Fanuc KAREL source: kd00015.KL

-- PROVISIONAL review KL for V940-1; original PC SHA256 e6e87a3893e7b443648327836266338668fe3b07deccfcc8bc3f06a5f374e33c
-- Incomplete behavior may be omitted. Consult companion uncertainty JSON. Do not deploy.
PROGRAM KD00015
%NOLOCKGROUP
VAR
  I : INTEGER
  J : INTEGER
  B : BOOLEAN
  R : REAL
  S : STRING[80]
BEGIN
  -- V9_ZERO_TABLE_METADATA_HINT layout=0001; no indexed target words; source/name/runtime held
  -- UNRESOLVED_PC offsets 5-6; opcodes 16
  -- UNRESOLVED_PC offsets 11-15; opcodes 7F
END KD00015
